Universal Robots PolyScope program: test.urp

Program test (installation=default directory=/programs createdIn=5.2.0.61336 lastSavedIn=5.2.0.61336 robotSerialNumber=20195500451)
Calibrated DH parameters: a=[0.00002, -0.231658, -0.317125, 0.000011, 0.000055, 0]; d=[0.162082, 123.190176, -180.284242, 57.22734, 0.099524, 0.09934]; alpha=[1.569304, 0.00289, 0.004025, 1.569925, -1.569026, 0]; deltaTheta=[0, 0.993923, 4.662183, 0.627072, 0.000001, 0]
Robot Program (runOnlyOnce=false)
  URCap 3F Gripper Activate (Robotiq_3-Finger_Adaptive_Gripper, Robotiq inc.) dataModel(r3factivate=1)
  URCap 3F Gripper Move (Robotiq_3-Finger_Adaptive_Gripper, Robotiq inc.) dataModel(speed=100, force=100, r3fwait=true, r3fmode=1, position=250)
  URCap 3F Gripper Move (Robotiq_3-Finger_Adaptive_Gripper, Robotiq inc.) dataModel(r3fwait=true, speed=100, force=100, position=0, r3fmode=1)
